PROGRAM Initialize
VAR
END_VAR

//*******************************************************
// SUBROUTINE Initialize
//*******************************************************
IF NOT SystemRunning THEN
    Step := 0;
    BottleCount := 0;
    CapCount := 0;
    Run_Bottle_Feeder := FALSE;
    Fill_Bottles_Solenoid := FALSE;
    Apply_Caps_Solenoid := FALSE;
    Push_Off_Bottles_Solenoid := FALSE;
END_IF

END_PROGRAM

(* stored: Version 1.1.0.1
   POU Initialize: Id {70163d09-83bf-43fc-b78c-35b24344d844}, SpecialFunc None *)
